// TIA Portal V16 export
// export: Created 2026-06-18T10:26:47.3066139Z, ExportSetting WithDefaults, DisplayName Totally Integrated Automation Portal, DisplayVersion V16 Update 8, DisplayName TIA Portal Version Control Interface, DisplayVersion V16 Update 8, DisplayName TIA Portal Openness, DisplayVersion V16 Update 8, DisplayName STEP 7 Professional, DisplayVersion V16 Update 8, DisplayName STEP 7 Safety, DisplayVersion V16 Update 7, DisplayName WinCC Professional, DisplayVersion V16 Update 8
Screen "Motor_Control"  800x480, Number=1
  ScreenLayer 
    IOField "IO_Speed" at 292,250 size 120x36  DataFormat=Decimal, FormatPattern=9999999, Mode=InOutput
    Button "BTN_Start" at 211,70 size 110x44  Mode=Text, TextOff="启动", TextOn="启动"
    Button "BTN_Reset" at 479,70 size 110x44  Mode=Text, TextOff="复位", TextOn="复位"
    Button "BTN_Stop" at 345,70 size 110x44  Mode=Text, TextOff="停止", TextOn="停止"
    SymbolicIOField "SIO_Mode" at 312,310 size 160x36  CountVisibleItems=3, Mode=InOutput, OnValue=1, TextOff="0", TextOn="1"
    Circle "LMP_Run" at 280,160 size 48x48
    Circle "LMP_Fault" at 400,160 size 48x48
    TextField "TXT_Title" at 200,20 size 400x32  Text="电机控制画面"
    TextField "TXT_ModeLabel" at 220,310 size 80x28  Text="运行模式"
    TextField "TXT_SpeedLabel" at 220,250 size 60x28  Text="转速"
